FUNCTION_BLOCK Switch_4P
VAR_INPUT
END_VAR
VAR_OUTPUT
END_VAR
VAR
	DIinput AT %I* : BOOL;
	DIinput2 AT %I* : BOOL;
	DIinput3 at %I* : bool;
END_VAR

PROPERTY Po0 : BOOL
GET
Po0 := not DIinput;
END_GET
END_PROPERTY

PROPERTY Po1 : BOOL
GET
Po1 := DIinput;
END_GET
END_PROPERTY

PROPERTY Po2 : BOOL
GET
Po2 := DIinput2;
END_GET
END_PROPERTY

PROPERTY Po3 : BOOL
GET
Po3 := DIinput3;
END_GET
END_PROPERTY

END_FUNCTION_BLOCK

(* stored: Version 1.1.0.1
   POU Switch_4P: Id {8f313100-a740-4dc6-a87a-fe2e594a95ab}, SpecialFunc None
   Property Po0: Id {ca128236-1627-466c-a5d6-2d7638026a03}
   Get Get: Id {0ec3e797-25e8-4c7e-ac5b-ad677de3cf95}
   Property Po1: Id {3d0d558c-89a2-4c2a-b09a-4ae0807c200a}
   Get Get: Id {5b787984-3882-43d6-9f7e-7b5ae6f56464}
   Property Po2: Id {5ed536d4-7e53-49e0-a670-789ccecff949}
   Get Get: Id {601d8eaa-b399-4d5d-95a0-7a4dbfd5161d}
   Property Po3: Id {434c0eb7-ff66-413f-ae69-eb50725fbbe8}
   Get Get: Id {cce7133e-a393-465e-9670-35d0ff4b26ad} *)
